FUNCTION IsNull : BOOL
VAR_INPUT
	anyPtrType		: ANY;
END_VAR

IF anyPtrType.diSize = SIZEOF(POINTER TO BYTE) THEN
	IsNull := anyPtrType.pValue^ = 0;
END_IF

END_FUNCTION

(* stored: Version 1.1.0.1
   POU IsNull: Id {fb608fd7-adb1-4f4b-830d-e41af9edea98}, SpecialFunc None *)
